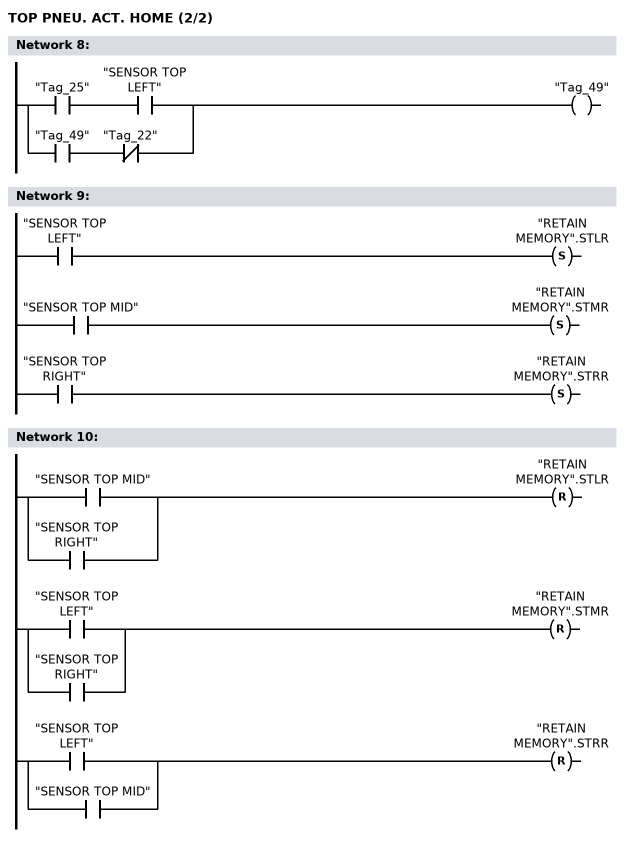
   RUNG wire#powerrail
      Contact( "Tag_25" )
      Contact( "SENSOR TOP LEFT" )
      wire#w1
      Coil( "Tag_49" )
   END_RUNG
   RUNG wire#powerrail
      Contact( "Tag_49" )
      I_Contact( "Tag_22" )
   END_RUNG wire#w1
   // the same network as SCL:
   "Tag_49" := ("Tag_25" AND "SENSOR TOP LEFT") OR ("Tag_49" AND NOT "Tag_22");
END_REGION

REGION Network 9
   RUNG wire#powerrail
      Contact( "SENSOR TOP LEFT" )
      S_Coil( "RETAIN MEMORY".STLR )
   END_RUNG
   RUNG wire#powerrail
      Contact( "SENSOR TOP MID" )
      S_Coil( "RETAIN MEMORY".STMR )
   END_RUNG
   RUNG wire#powerrail
      Contact( "SENSOR TOP RIGHT" )
      S_Coil( "RETAIN MEMORY".STRR )
   END_RUNG
   // the same network as SCL:
   IF "SENSOR TOP LEFT" THEN "RETAIN MEMORY".STLR := TRUE; END_IF;
   IF "SENSOR TOP MID" THEN "RETAIN MEMORY".STMR := TRUE; END_IF;
   IF "SENSOR TOP RIGHT" THEN "RETAIN MEMORY".STRR := TRUE; END_IF;
END_REGION

REGION Network 10
   RUNG wire#powerrail
      Contact( "SENSOR TOP MID" )
      wire#w1
      R_Coil( "RETAIN MEMORY".STLR )
   END_RUNG
   RUNG wire#powerrail
      Contact( "SENSOR TOP RIGHT" )
   END_RUNG wire#w1
   RUNG wire#powerrail
      Contact( "SENSOR TOP LEFT" )
      wire#w2
      R_Coil( "RETAIN MEMORY".STMR )
   END_RUNG
   RUNG wire#powerrail
      Contact( "SENSOR TOP RIGHT" )
   END_RUNG wire#w2
   RUNG wire#powerrail
      Contact( "SENSOR TOP LEFT" )
      wire#w3
      R_Coil( "RETAIN MEMORY".STRR )
   END_RUNG
   RUNG wire#powerrail
      Contact( "SENSOR TOP MID" )
   END_RUNG wire#w3
   // the same network as SCL:
   IF "SENSOR TOP MID" OR "SENSOR TOP RIGHT" THEN "RETAIN MEMORY".STLR := FALSE; END_IF;
   IF "SENSOR TOP LEFT" OR "SENSOR TOP RIGHT" THEN "RETAIN MEMORY".STMR := FALSE; END_IF;
   IF "SENSOR TOP LEFT" OR "SENSOR TOP MID" THEN "RETAIN MEMORY".STRR := FALSE; END_IF;
END_REGION
END_FUNCTION

FUNCTION "TOP PNEU. ACT. AUTO" : Void   // FC11, LAD
{ S7_Optimized_Access := 'TRUE' }
VERSION : 0.1
BEGIN

REGION Network 1
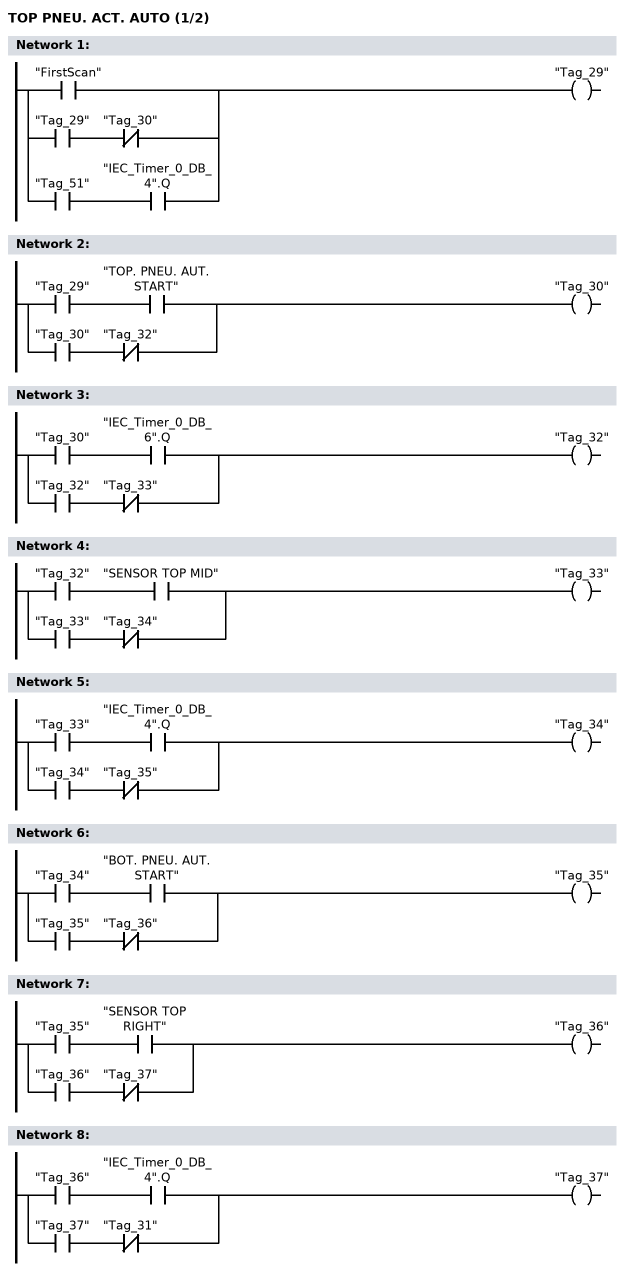
   RUNG wire#powerrail
      Contact( "FirstScan" )
      wire#w1
      Coil( "Tag_29" )
   END_RUNG
   RUNG wire#powerrail
      Contact( "Tag_29" )
      I_Contact( "Tag_30" )
   END_RUNG wire#w1
   RUNG wire#powerrail
      Contact( "Tag_51" )
      Contact( "IEC_Timer_0_DB_4".Q )
   END_RUNG wire#w1
   // the same network as SCL:
   "Tag_29" := "FirstScan" OR ("Tag_29" AND NOT "Tag_30") OR ("Tag_51" AND "IEC_Timer_0_DB_4".Q);
END_REGION

REGION Network 2
   RUNG wire#powerrail
      Contact( "Tag_29" )
      Contact( "TOP. PNEU. AUT. START" )
      wire#w1
      Coil( "Tag_30" )
   END_RUNG
   RUNG wire#powerrail
      Contact( "Tag_30" )
      I_Contact( "Tag_32" )
   END_RUNG wire#w1
   // the same network as SCL:
   "Tag_30" := ("Tag_29" AND "TOP. PNEU. AUT. START") OR ("Tag_30" AND NOT "Tag_32");
END_REGION

REGION Network 3
   RUNG wire#powerrail
      Contact( "Tag_30" )
      Contact( "IEC_Timer_0_DB_6".Q )
      wire#w1
      Coil( "Tag_32" )
   END_RUNG
   RUNG wire#powerrail
      Contact( "Tag_32" )
      I_Contact( "Tag_33" )
   END_RUNG wire#w1
   // the same network as SCL:
   "Tag_32" := ("Tag_30" AND "IEC_Timer_0_DB_6".Q) OR ("Tag_32" AND NOT "Tag_33");
END_REGION

REGION Network 4
   RUNG wire#powerrail
      Contact( "Tag_32" )
      Contact( "SENSOR TOP MID" )
      wire#w1
      Coil( "Tag_33" )
   END_RUNG
   RUNG wire#powerrail
      Contact( "Tag_33" )
      I_Contact( "Tag_34" )
   END_RUNG wire#w1
   // the same network as SCL:
   "Tag_33" := ("Tag_32" AND "SENSOR TOP MID") OR ("Tag_33" AND NOT "Tag_34");
END_REGION

REGION Network 5
   RUNG wire#powerrail
      Contact( "Tag_33" )
      Contact( "IEC_Timer_0_DB_4".Q )
      wire#w1
      Coil( "Tag_34" )
   END_RUNG
   RUNG wire#powerrail
      Contact( "Tag_34" )
      I_Contact( "Tag_35" )
   END_RUNG wire#w1
   // the same network as SCL:
   "Tag_34" := ("Tag_33" AND "IEC_Timer_0_DB_4".Q) OR ("Tag_34" AND NOT "Tag_35");
END_REGION

REGION Network 6
   RUNG wire#powerrail
      Contact( "Tag_34" )
      Contact( "BOT. PNEU. AUT. START" )
      wire#w1
      Coil( "Tag_35" )
   END_RUNG
   RUNG wire#powerrail
      Contact( "Tag_35" )
      I_Contact( "Tag_36" )
   END_RUNG wire#w1
   // the same network as SCL:
   "Tag_35" := ("Tag_34" AND "BOT. PNEU. AUT. START") OR ("Tag_35" AND NOT "Tag_36");
END_REGION

REGION Network 7
   RUNG wire#powerrail
      Contact( "Tag_35" )
      Contact( "SENSOR TOP RIGHT" )
      wire#w1
      Coil( "Tag_36" )
   END_RUNG
   RUNG wire#powerrail
      Contact( "Tag_36" )
      I_Contact( "Tag_37" )
   END_RUNG wire#w1
   // the same network as SCL:
   "Tag_36" := ("Tag_35" AND "SENSOR TOP RIGHT") OR ("Tag_36" AND NOT "Tag_37");
END_REGION

REGION Network 8
   RUNG wire#powerrail
      Contact( "Tag_36" )
      Contact( "IEC_Timer_0_DB_4".Q )
      wire#w1
      Coil( "Tag_37" )
   END_RUNG
   RUNG wire#powerrail
      Contact( "Tag_37" )
      I_Contact( "Tag_31" )
   END_RUNG wire#w1
   // the same network as SCL:
   "Tag_37" := ("Tag_36" AND "IEC_Timer_0_DB_4".Q) OR ("Tag_37" AND NOT "Tag_31");
END_REGION

REGION Network 9
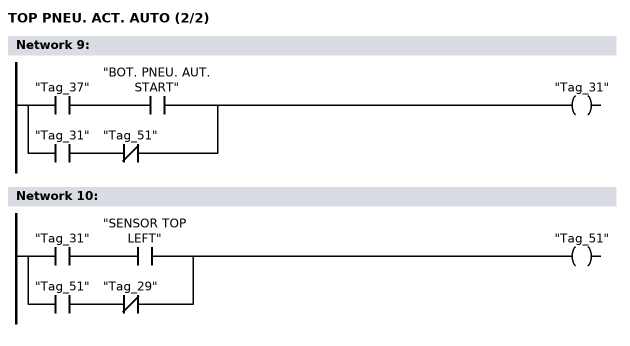
   RUNG wire#powerrail
      Contact( "Tag_37" )
      Contact( "BOT. PNEU. AUT. START" )
      wire#w1
      Coil( "Tag_31" )
   END_RUNG
   RUNG wire#powerrail
      Contact( "Tag_31" )
      I_Contact( "Tag_51" )
   END_RUNG wire#w1
   // the same network as SCL:
   "Tag_31" := ("Tag_37" AND "BOT. PNEU. AUT. START") OR ("Tag_31" AND NOT "Tag_51");
END_REGION

REGION Network 10
   RUNG wire#powerrail
      Contact( "Tag_31" )
      Contact( "SENSOR TOP LEFT" )
      wire#w1
      Coil( "Tag_51" )
   END_RUNG
   RUNG wire#powerrail
      Contact( "Tag_51" )
      I_Contact( "Tag_29" )
   END_RUNG wire#w1
   // the same network as SCL:
   "Tag_51" := ("Tag_31" AND "SENSOR TOP LEFT") OR ("Tag_51" AND NOT "Tag_29");
END_REGION
END_FUNCTION

FUNCTION "VERT. PNEU. ACT. HOME" : Void   // FC12, LAD
{ S7_Optimized_Access := 'TRUE' }
VERSION : 0.1
BEGIN

REGION Network 1
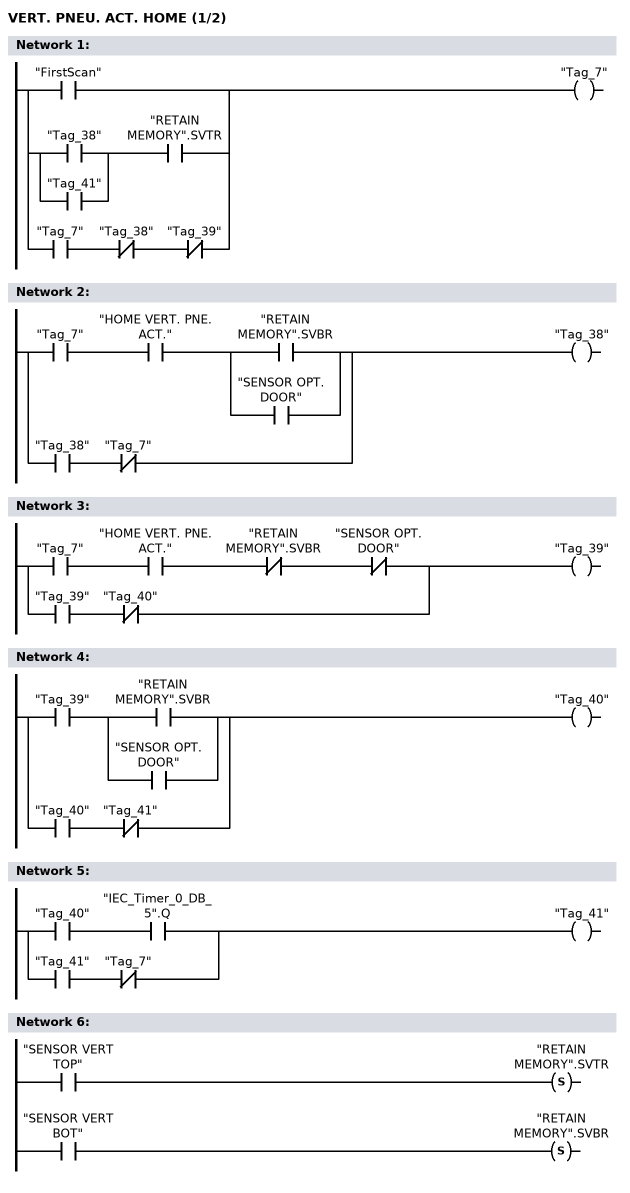
   RUNG wire#powerrail
      Contact( "FirstScan" )
      wire#w1
      Coil( "Tag_7" )
   END_RUNG
   RUNG wire#powerrail
      Contact( "Tag_38" )
      wire#w2
      Contact( "RETAIN MEMORY".SVTR )
   END_RUNG wire#w1
   RUNG wire#powerrail
      Contact( "Tag_41" )
   END_RUNG wire#w2
   RUNG wire#powerrail
      Contact( "Tag_7" )
      I_Contact( "Tag_38" )
      I_Contact( "Tag_39" )
   END_RUNG wire#w1
   // the same network as SCL:
   "Tag_7" := "FirstScan" OR (("Tag_38" OR "Tag_41") AND "RETAIN MEMORY".SVTR) OR ("Tag_7" AND NOT "Tag_38" AND NOT "Tag_39");
END_REGION

REGION Network 2
   RUNG wire#powerrail
      Contact( "Tag_7" )
      Contact( "HOME VERT. PNE. ACT." )
      wire#w1
      Contact( "RETAIN MEMORY".SVBR )
      wire#w2
      Coil( "Tag_38" )
   END_RUNG
   RUNG wire#w1
      Contact( "SENSOR OPT. DOOR" )
   END_RUNG wire#w2
   RUNG wire#powerrail
      Contact( "Tag_38" )
      I_Contact( "Tag_7" )
   END_RUNG wire#w2
   // the same network as SCL:
   "Tag_38" := ("Tag_7" AND "HOME VERT. PNE. ACT." AND ("RETAIN MEMORY".SVBR OR "SENSOR OPT. DOOR")) OR ("Tag_38" AND NOT "Tag_7");
END_REGION

REGION Network 3
   RUNG wire#powerrail
      Contact( "Tag_7" )
      Contact( "HOME VERT. PNE. ACT." )
      I_Contact( "RETAIN MEMORY".SVBR )
      I_Contact( "SENSOR OPT. DOOR" )
      wire#w1
      Coil( "Tag_39" )
   END_RUNG
   RUNG wire#powerrail
      Contact( "Tag_39" )
      I_Contact( "Tag_40" )
   END_RUNG wire#w1
   // the same network as SCL:
   "Tag_39" := ("Tag_7" AND "HOME VERT. PNE. ACT." AND NOT "RETAIN MEMORY".SVBR AND NOT "SENSOR OPT. DOOR") OR ("Tag_39" AND NOT "Tag_40");
END_REGION

REGION Network 4
   RUNG wire#powerrail
      Contact( "Tag_39" )
      wire#w1
      Contact( "RETAIN MEMORY".SVBR )
      wire#w2
      Coil( "Tag_40" )
   END_RUNG
   RUNG wire#w1
      Contact( "SENSOR OPT. DOOR" )
   END_RUNG wire#w2
   RUNG wire#powerrail
      Contact( "Tag_40" )
      I_Contact( "Tag_41" )
   END_RUNG wire#w2
   // the same network as SCL:
   "Tag_40" := ("Tag_39" AND ("RETAIN MEMORY".SVBR OR "SENSOR OPT. DOOR")) OR ("Tag_40" AND NOT "Tag_41");
END_REGION

REGION Network 5
   RUNG wire#powerrail
      Contact( "Tag_40" )
      Contact( "IEC_Timer_0_DB_5".Q )
      wire#w1
      Coil( "Tag_41" )
   END_RUNG
   RUNG wire#powerrail
      Contact( "Tag_41" )
      I_Contact( "Tag_7" )
   END_RUNG wire#w1
   // the same network as SCL:
   "Tag_41" := ("Tag_40" AND "IEC_Timer_0_DB_5".Q) OR ("Tag_41" AND NOT "Tag_7");
END_REGION

REGION Network 6
   RUNG wire#powerrail
      Contact( "SENSOR VERT TOP" )
      S_Coil( "RETAIN MEMORY".SVTR )
   END_RUNG
   RUNG wire#powerrail
      Contact( "SENSOR VERT BOT" )
      S_Coil( "RETAIN MEMORY".SVBR )
   END_RUNG
   // the same network as SCL:
   IF "SENSOR VERT TOP" THEN "RETAIN MEMORY".SVTR := TRUE; END_IF;
   IF "SENSOR VERT BOT" THEN "RETAIN MEMORY".SVBR := TRUE; END_IF;
END_REGION

REGION Network 7
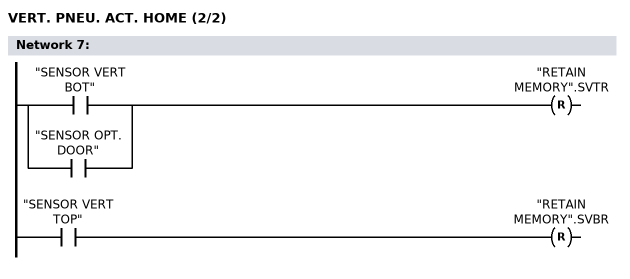
   RUNG wire#powerrail
      Contact( "SENSOR VERT BOT" )
      wire#w1
      R_Coil( "RETAIN MEMORY".SVTR )
   END_RUNG
   RUNG wire#powerrail
      Contact( "SENSOR OPT. DOOR" )
   END_RUNG wire#w1
   RUNG wire#powerrail
      Contact( "SENSOR VERT TOP" )
      R_Coil( "RETAIN MEMORY".SVBR )
   END_RUNG
   // the same network as SCL:
   IF "SENSOR VERT BOT" OR "SENSOR OPT. DOOR" THEN "RETAIN MEMORY".SVTR := FALSE; END_IF;
   IF "SENSOR VERT TOP" THEN "RETAIN MEMORY".SVBR := FALSE; END_IF;
END_REGION
END_FUNCTION

FUNCTION "VERT. PNEU. ACT. AUTO" : Void   // FC13, LAD
{ S7_Optimized_Access := 'TRUE' }
VERSION : 0.1
BEGIN

REGION Network 1
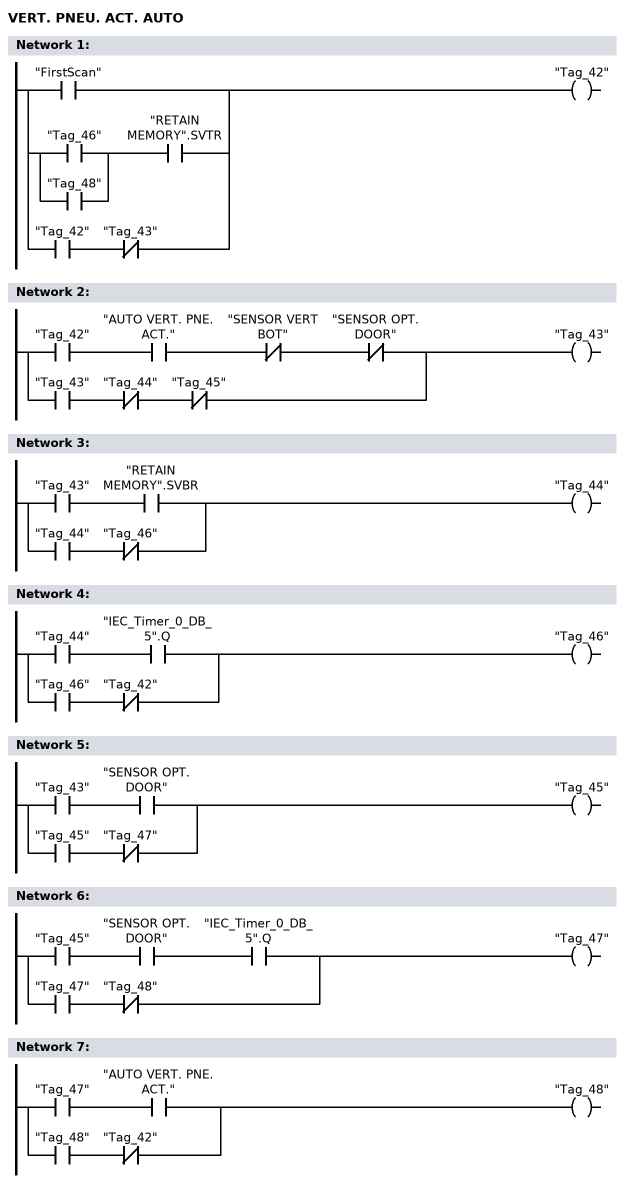
   RUNG wire#powerrail
      Contact( "FirstScan" )
      wire#w1
      Coil( "Tag_42" )
   END_RUNG
   RUNG wire#powerrail
      Contact( "Tag_46" )
      wire#w2
      Contact( "RETAIN MEMORY".SVTR )
   END_RUNG wire#w1
   RUNG wire#powerrail
      Contact( "Tag_48" )
   END_RUNG wire#w2
   RUNG wire#powerrail
      Contact( "Tag_42" )
      I_Contact( "Tag_43" )
   END_RUNG wire#w1
   // the same network as SCL:
   "Tag_42" := "FirstScan" OR (("Tag_46" OR "Tag_48") AND "RETAIN MEMORY".SVTR) OR ("Tag_42" AND NOT "Tag_43");
END_REGION

REGION Network 2
   RUNG wire#powerrail
      Contact( "Tag_42" )
      Contact( "AUTO VERT. PNE. ACT." )
      I_Contact( "SENSOR VERT BOT" )
      I_Contact( "SENSOR OPT. DOOR" )
      wire#w1
      Coil( "Tag_43" )
   END_RUNG
   RUNG wire#powerrail
      Contact( "Tag_43" )
      I_Contact( "Tag_44" )
      I_Contact( "Tag_45" )
   END_RUNG wire#w1
   // the same network as SCL:
   "Tag_43" := ("Tag_42" AND "AUTO VERT. PNE. ACT." AND NOT "SENSOR VERT BOT" AND NOT "SENSOR OPT. DOOR") OR ("Tag_43" AND NOT "Tag_44" AND NOT "Tag_45");
END_REGION

REGION Network 3
   RUNG wire#powerrail
      Contact( "Tag_43" )
      Contact( "RETAIN MEMORY".SVBR )
      wire#w1
      Coil( "Tag_44" )
   END_RUNG
   RUNG wire#powerrail
      Contact( "Tag_44" )
      I_Contact( "Tag_46" )
   END_RUNG wire#w1
   // the same network as SCL:
   "Tag_44" := ("Tag_43" AND "RETAIN MEMORY".SVBR) OR ("Tag_44" AND NOT "Tag_46");
END_REGION

REGION Network 4
   RUNG wire#powerrail
      Contact( "Tag_44" )
      Contact( "IEC_Timer_0_DB_5".Q )
      wire#w1
      Coil( "Tag_46" )
   END_RUNG
   RUNG wire#powerrail
      Contact( "Tag_46" )
      I_Contact( "Tag_42" )
   END_RUNG wire#w1
   // the same network as SCL:
   "Tag_46" := ("Tag_44" AND "IEC_Timer_0_DB_5".Q) OR ("Tag_46" AND NOT "Tag_42");
END_REGION

REGION Network 5
   RUNG wire#powerrail
      Contact( "Tag_43" )
      Contact( "SENSOR OPT. DOOR" )
      wire#w1
      Coil( "Tag_45" )
   END_RUNG
   RUNG wire#powerrail
      Contact( "Tag_45" )
      I_Contact( "Tag_47" )
   END_RUNG wire#w1
   // the same network as SCL:
   "Tag_45" := ("Tag_43" AND "SENSOR OPT. DOOR") OR ("Tag_45" AND NOT "Tag_47");
END_REGION

REGION Network 6
   RUNG wire#powerrail
      Contact( "Tag_45" )
      Contact( "SENSOR OPT. DOOR" )
      Contact( "IEC_Timer_0_DB_5".Q )
      wire#w1
      Coil( "Tag_47" )
   END_RUNG
   RUNG wire#powerrail
      Contact( "Tag_47" )
      I_Contact( "Tag_48" )
   END_RUNG wire#w1
   // the same network as SCL:
   "Tag_47" := ("Tag_45" AND "SENSOR OPT. DOOR" AND "IEC_Timer_0_DB_5".Q) OR ("Tag_47" AND NOT "Tag_48");
END_REGION

REGION Network 7
   RUNG wire#powerrail
      Contact( "Tag_47" )
      Contact( "AUTO VERT. PNE. ACT." )
      wire#w1
      Coil( "Tag_48" )
   END_RUNG
   RUNG wire#powerrail
      Contact( "Tag_48" )
      I_Contact( "Tag_42" )
   END_RUNG wire#w1
   // the same network as SCL:
   "Tag_48" := ("Tag_47" AND "AUTO VERT. PNE. ACT.") OR ("Tag_48" AND NOT "Tag_42");
END_REGION
END_FUNCTION

ORGANIZATION_BLOCK "MAIN"   // OB1, LAD, ProgramCycle
TITLE = "Main Program Sweep (Cycle)"
{ S7_Optimized_Access := 'TRUE' }
VERSION : 0.1
   VAR_INPUT
      Initial_Call : Bool;   // Initial call of this OB
      Remanence : Bool;   // =True, if remanent data are available
   END_VAR
   VAR_TEMP   // added for the SCL form of the ladder/FBD networks
      _w1 : Bool;
   END_VAR
BEGIN

REGION Network 1
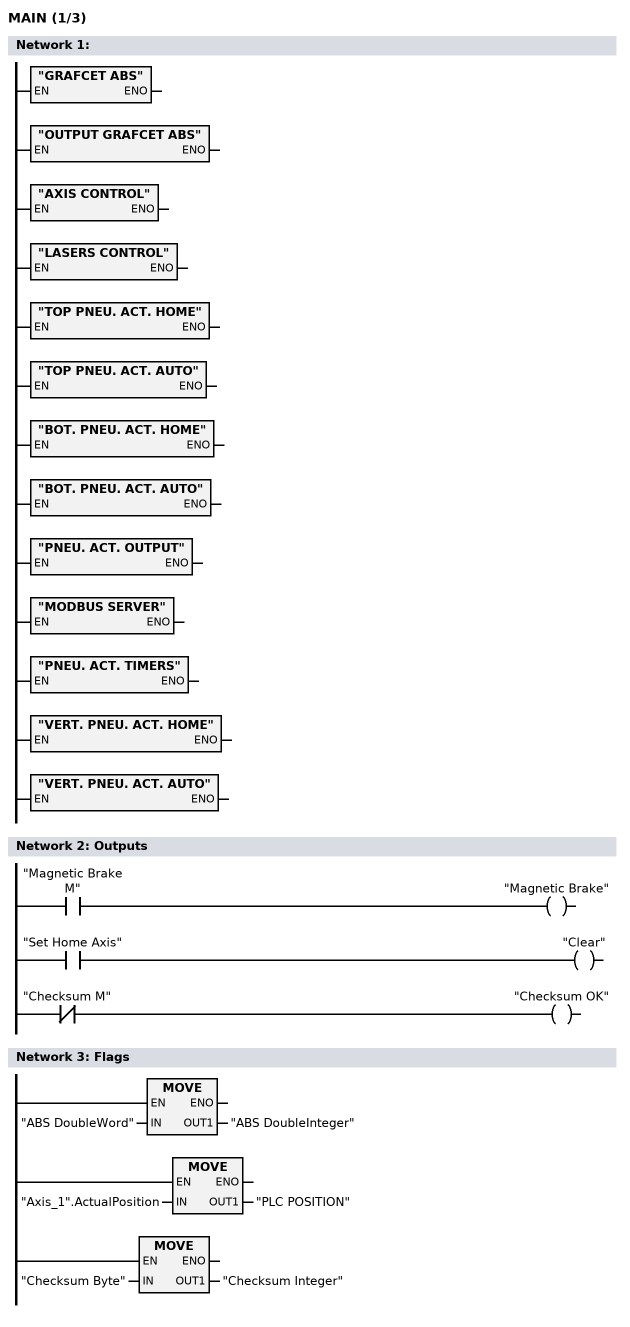
   RUNG wire#powerrail
      "GRAFCET ABS"()
   END_RUNG
   RUNG wire#powerrail
      "OUTPUT GRAFCET ABS"()
   END_RUNG
   RUNG wire#powerrail
      "AXIS CONTROL"()
   END_RUNG
   RUNG wire#powerrail
      "LASERS CONTROL"()
   END_RUNG
   RUNG wire#powerrail
      "TOP PNEU. ACT. HOME"()
   END_RUNG
   RUNG wire#powerrail
      "TOP PNEU. ACT. AUTO"()
   END_RUNG
   RUNG wire#powerrail
      "BOT. PNEU. ACT. HOME"()
   END_RUNG
   RUNG wire#powerrail
      "BOT. PNEU. ACT. AUTO"()
   END_RUNG
   RUNG wire#powerrail
      "PNEU. ACT. OUTPUT"()
   END_RUNG
   RUNG wire#powerrail
      "MODBUS SERVER"()
   END_RUNG
   RUNG wire#powerrail
      "PNEU. ACT. TIMERS"()
   END_RUNG
   RUNG wire#powerrail
      "VERT. PNEU. ACT. HOME"()
   END_RUNG
   RUNG wire#powerrail
      "VERT. PNEU. ACT. AUTO"()
   END_RUNG
   // the same network as SCL:
   "GRAFCET ABS"();
   "OUTPUT GRAFCET ABS"();
   "AXIS CONTROL"();
   "LASERS CONTROL"();
   "TOP PNEU. ACT. HOME"();
   "TOP PNEU. ACT. AUTO"();
   "BOT. PNEU. ACT. HOME"();
   "BOT. PNEU. ACT. AUTO"();
   "PNEU. ACT. OUTPUT"();
   "MODBUS SERVER"();
   "PNEU. ACT. TIMERS"();
   "VERT. PNEU. ACT. HOME"();
   "VERT. PNEU. ACT. AUTO"();
END_REGION

REGION Network 2: Outputs
   RUNG wire#powerrail
      Contact( "Magnetic Brake M" )
      Coil( "Magnetic Brake" )
   END_RUNG
   RUNG wire#powerrail
      Contact( "Set Home Axis" )
      Coil( "Clear" )
   END_RUNG
   RUNG wire#powerrail
      I_Contact( "Checksum M" )
      Coil( "Checksum OK" )
   END_RUNG
   // the same network as SCL:
   "Magnetic Brake" := "Magnetic Brake M";
   "Clear" := "Set Home Axis";
   "Checksum OK" := NOT "Checksum M";
END_REGION

REGION Network 3: Flags
   RUNG wire#powerrail
      Move(in := "ABS DoubleWord", out1 => "ABS DoubleInteger")
   END_RUNG
   RUNG wire#powerrail
      Move(in := "Axis_1".ActualPosition, out1 => "PLC POSITION")
   END_RUNG
   RUNG wire#powerrail
      Move(in := "Checksum Byte", out1 => "Checksum Integer")
   END_RUNG
   // the same network as SCL:
   "ABS DoubleInteger" := "ABS DoubleWord";
   "PLC POSITION" := "Axis_1".ActualPosition;
   "Checksum Integer" := "Checksum Byte";
END_REGION

REGION Network 4
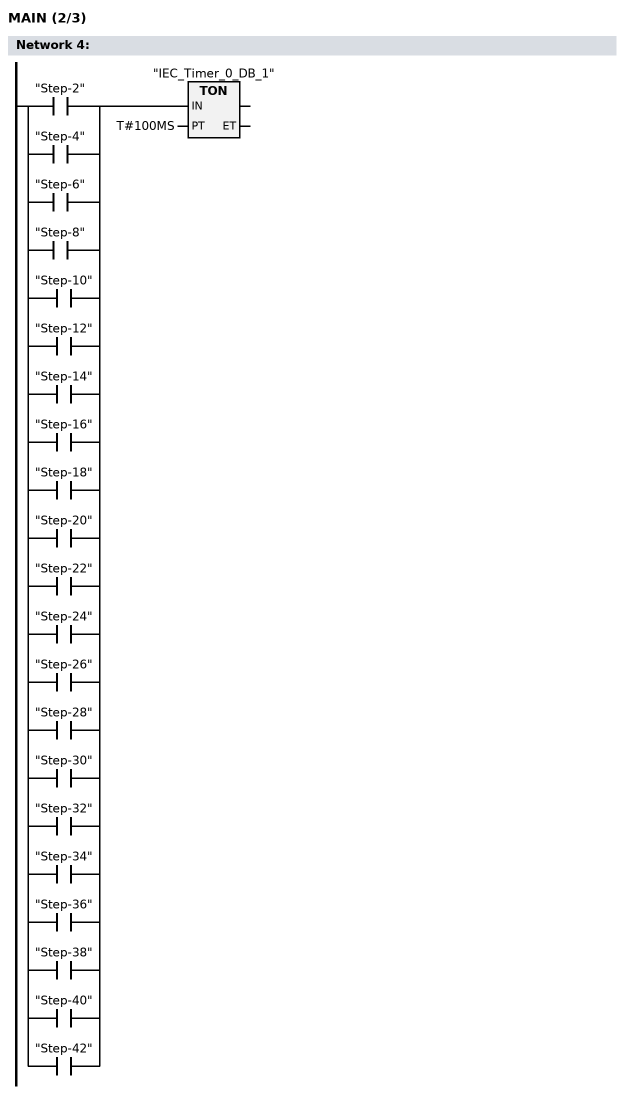
   "IEC_Timer_0_DB_1".TON(IN := "Step-2" OR "Step-4" OR "Step-6" OR "Step-8" OR "Step-10" OR "Step-12" OR "Step-14" OR "Step-16" OR "Step-18" OR "Step-20" OR "Step-22" OR "Step-24" OR "Step-26" OR "Step-28" OR "Step-30" OR "Step-32" OR "Step-34" OR "Step-36" OR "Step-38" OR "Step-40" OR "Step-42",
                          PT := T#100MS);
END_REGION

REGION Network 5
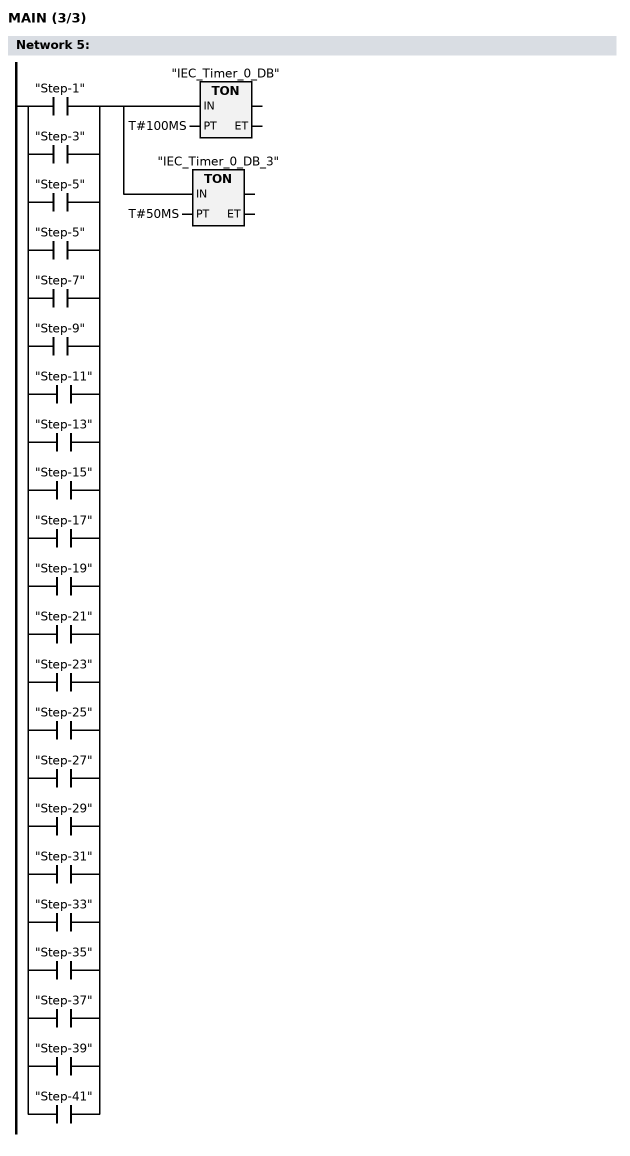
   #_w1 := "Step-1" OR "Step-3" OR "Step-5" OR "Step-5" OR "Step-7" OR "Step-9" OR "Step-11" OR "Step-13" OR "Step-15" OR "Step-17" OR "Step-19" OR "Step-21" OR "Step-23" OR "Step-25" OR "Step-27" OR "Step-29" OR "Step-31" OR "Step-33" OR "Step-35" OR "Step-37" OR "Step-39" OR "Step-41";
   "IEC_Timer_0_DB".TON(IN := #_w1, PT := T#100MS);
   "IEC_Timer_0_DB_3".TON(IN := #_w1, PT := T#50MS);
END_REGION
END_ORGANIZATION_BLOCK